TYPE ST_Data_PRR :
STRUCT
	pump		:DINT;
	stage		:STRING;
	rinse1		:REAL;
	rinse2		:REAL;
	wash1		:REAL;
	wash2		:REAL;
	
END_STRUCT
END_TYPE

(* stored: Version 1.1.0.1, ProductVersion 3.1.4024.12
   DUT ST_Data_PRR: Id {9a320d08-c4f3-4f03-b79e-7af5e24f6ea4} *)
